// TIA Portal V18 export
TYPE "LGasp_Type_packetdata"
// stored: IsFailsafeCompliant false
   STRUCT
      lunghezza : Real;   // lunghezza del pezzo
      IDERP : DInt;   // dato 210100085
      ID : DInt;   // ID riga della pagina di produzione
   END_STRUCT;
END_TYPE
